(* Logix 5000 project; controller Torque_Testing vendor 1 type 14 code 196 rev 32.14; software revision 32.05 *)

TASK MainTask (continuous, watchdog 500 ms) : MainProgram

MODULES
   Local : vendor 1 type 14 code 196 (5069 0, rev 32.14)
      Torque_Testing : ETHERNET-MODULE (Ethernet 10.138.27.3, rev 1.1, Output RPI 10 ms)
END_MODULES

PROGRAM MainProgram   (* main routine MainRoutine *)

ROUTINE MainRoutine   (* ladder *)
END_ROUTINE
END_PROGRAM
